{attribute 'GeneratedUsingTerminal: EL2212-0000-0020'}
{attribute addProperty BoxType "EL2212-0000-0020"}
{attribute addProperty Id "Ready_to_activateBOOL1Output_activeBOOL1Tristate_activeBOOL1PWM_activeBOOL1WarningBOOL1ErrorBOOL1TxPDO_ToggleBOOL1"}
{attribute addProperty CRC "2369768739"}
{attribute addProperty Size "7"}
TYPE Status_8D3FCD23 :
STRUCT
	{attribute addProperty Name "Ready_to_activate"}
	Ready_to_activate : BOOL;
	{attribute addProperty Name "Output_active"}
	Output_active : BOOL;
	{attribute addProperty Name "Tristate_active"}
	Tristate_active : BOOL;
	{attribute addProperty Name "PWM_active"}
	PWM_active : BOOL;
	{attribute addProperty Name "Warning"}
	Warning : BOOL;
	{attribute addProperty Name "Error"}
	Error : BOOL;
	{attribute addProperty Name "TxPDO_Toggle"}
	TxPDO_Toggle : BOOL;
END_STRUCT
END_TYPE

(* stored: Version 1.2.0.0, ProductVersion 3.1.4024.9
   DUT Status_8D3FCD23: Id {b68ce937-354b-4d04-b73a-0e845968d675} *)
